FUNCTION_BLOCK FB_IOManager
VAR_INPUT
END_VAR
VAR_OUTPUT
END_VAR
VAR
	fbAI 	:	FB_Analogin;
	fbAO	:	FB_AnalogOut;
	fbDI	:	FB_DigitalIn;
	fbDO	:	FB_DigitalOut;
	fbTC	:	FB_TCIn;
END_VAR

(*
fbAI(iMaxInCH	:=	HMI.iEnabledChannels_AI);
fbAO(iMaxInCH	:=	HMI.iEnabledChannels_AO);
fbDI(iMaxInCH	:=	HMI.iEnabledChannels_DI);
fbDO(iMaxInCH	:=	HMI.iEnabledChannels_DO);
fbTC(iMaxInCH	:=	HMI.iEnabledChannels_TC);
*)

fbAI(iMaxInCH	:=	6);
fbAO(iMaxInCH	:=	3);
fbDI(iMaxInCH	:=	30);
fbDO(iMaxInCH	:=	16);
fbTC(iMaxInCH	:=	12);

END_FUNCTION_BLOCK

(* stored: Version 1.1.0.1, ProductVersion 3.1.4024.12
   POU FB_IOManager: Id {edc8b196-c64d-442f-ac3e-65ea59a3ee6a}, SpecialFunc None *)
